Fanuc KAREL source: kt00895.KL

PROGRAM KT00895
%NOLOCKGROUP
VAR
P1 : XYZWPREXT;P2 : XYZWPREXT;OUT:BOOLEAN
BEGIN
--
--
P1.X=1.0
P2.Y=2.0
P1.X=1.0
P2.Y=2.0
OUT=IN_RANGE(P1)
END KT00895
